(* Logix 5000 project; controller IOL_Sample vendor 1 type 14 code 196 rev 30.11; software revision 30.02; part 7 of 7 *)

TYPE Generic_16_Words :
STRUCT
   Data : INT[16];
END_STRUCT
END_TYPE

TYPE Generic_28_Bytes :
STRUCT
   Data : SINT[28];
END_STRUCT
END_TYPE

ADD_ON_INSTRUCTION Turck_TN_Q40   (* revision 1.0 *)
VAR_IN_OUT
   Process_Data_In : Generic_16_Words; {required}
   Process_Data_Out : Generic_16_Words; {required}
END_VAR
VAR_OUTPUT
   Ready_Flag : BOOL; {visible}   // 1 -> 0 or 0 -> 1: Command executed, new data available 0 or 1: No new data available
   Error : BOOL; {visible}   // 0: Command executed error-free 1: Command executed with error
   Tag : BOOL; {visible}   // 0: No tag within the detection range 1: Tag present at read/write head
   Antenna_State : BOOL; {visible}   // 0: RF field switched off 1: RF field switched on
   CMDCPY : SINT; {visible}   // Command Code Echo
   Error_Code : SINT; {visible}   // Error Code (Check Manual)
   ALR2 : BOOL; {visible}   // 0: Alarm 2 off 1: Alarm 2 on
   ALR1 : BOOL; {visible}   // 0: Alarm 1 off 1: Alarm 1 on
   Address : SINT; {visible}   // Address of the first memory block on the tag on which a command was executed
   RSSI : SINT; {visible}   // Signal Strength
END_VAR
VAR_IN_OUT
   Read_Data : Generic_28_Bytes; {required}   // Data read from Tag
END_VAR
VAR_INPUT
   Start : BOOL; {visible}   // 1 -> 0 or 0 -> 1: Execute command. The START bit switches status automatically with the automatic read and automatic write commands. 0 or 1: Idle
   N_Ant : BOOL; {visible}   // 0: Switch on RF field 1: Switch off RF field
   CMD : SINT; {visible}   // 0: No command 1: Automatic read 2: Automatic write 3: Read 4: Write 5: Display UID and time stamp
   NB_Block : SINT; {visible}   // Number of memory blocks to be read or written n EEPROM: max. 7 memory blocks n FRAM: max. 3 memory blocks
   Start_Address : INT; {visible}   // Address of the first memory block on the tag on which a command is to be executed
END_VAR
VAR_IN_OUT
   Write_Data : Generic_28_Bytes; {required}   // Data to write to Tag
END_VAR

ROUTINE Logic   (* ladder *)
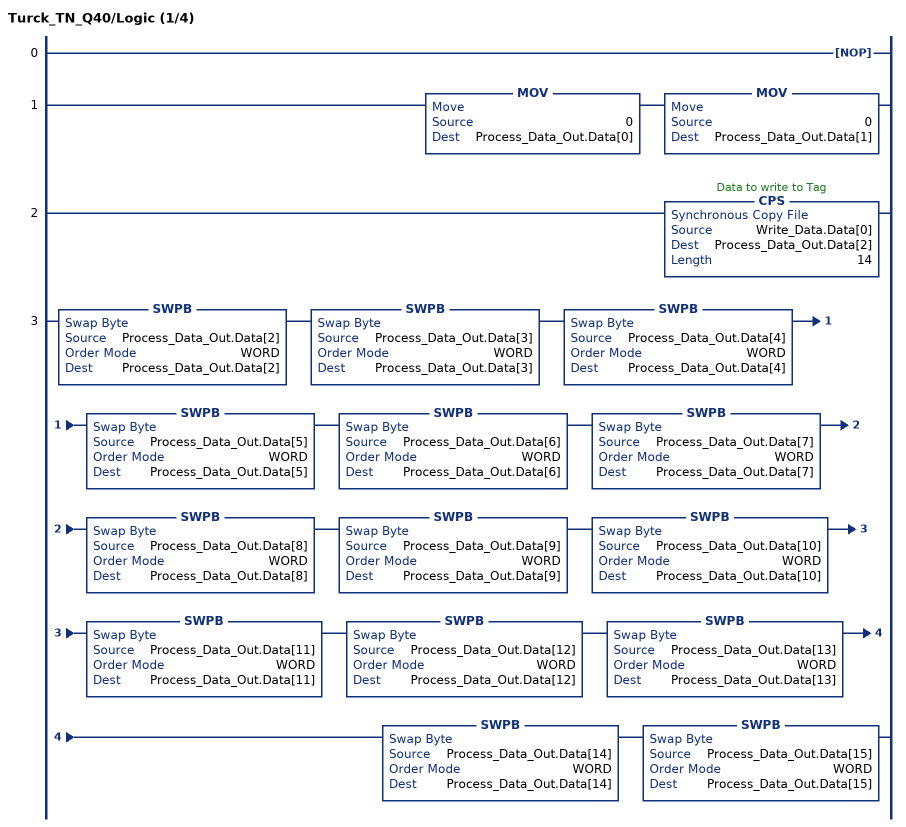
   0: NOP();
   1: MOV(0,Process_Data_Out.Data[0])MOV(0,Process_Data_Out.Data[1]);
   2: CPS(Write_Data.Data[0],Process_Data_Out.Data[2],14);
   3: SWPB(Process_Data_Out.Data[2],WORD,Process_Data_Out.Data[2])SWPB(Process_Data_Out.Data[3],WORD,Process_Data_Out.Data[3])SWPB(Process_Data_Out.Data[4],WORD,Process_Data_Out.Data[4])SWPB(Process_Data_Out.Data[5],WORD,Process_Data_Out.Data[5])SWPB(Process_Data_Out.Data[6],WORD,Process_Data_Out.Data[6])SWPB(Process_Data_Out.Data[7],WORD,Process_Data_Out.Data[7])SWPB(Process_Data_Out.Data[8],WORD,Process_Data_Out.Data[8])SWPB(Process_Data_Out.Data[9],WORD,Process_Data_Out.Data[9])SWPB(Process_Data_Out.Data[10],WORD,Process_Data_Out.Data[10])SWPB(Process_Data_Out.Data[11],WORD,Process_Data_Out.Data[11])SWPB(Process_Data_Out.Data[12],WORD,Process_Data_Out.Data[12])SWPB(Process_Data_Out.Data[13],WORD,Process_Data_Out.Data[13])SWPB(Process_Data_Out.Data[14],WORD,Process_Data_Out.Data[14])SWPB(Process_Data_Out.Data[15],WORD,Process_Data_Out.Data[15]);
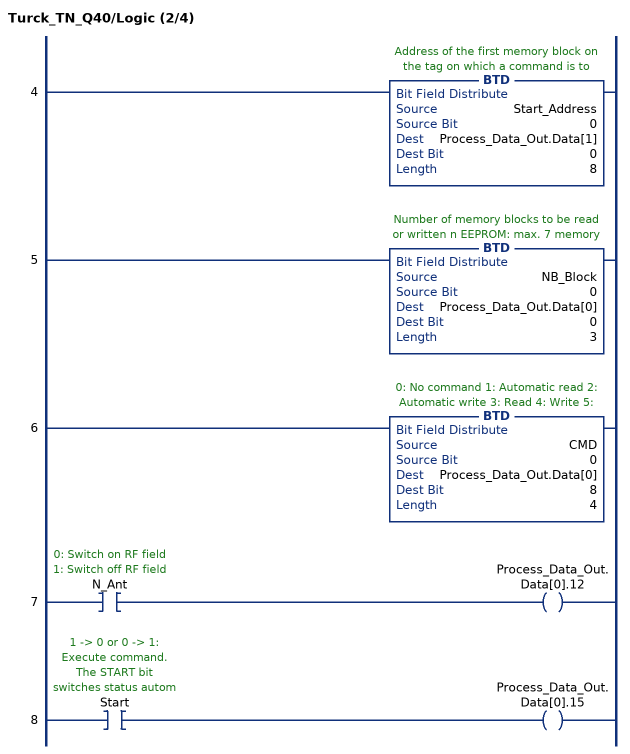
   4: BTD(Start_Address,0,Process_Data_Out.Data[1],0,8);
   5: BTD(NB_Block,0,Process_Data_Out.Data[0],0,3);
   6: BTD(CMD,0,Process_Data_Out.Data[0],8,4);
   7: XIC(N_Ant)OTE(Process_Data_Out.Data[0].12);
   8: XIC(Start)OTE(Process_Data_Out.Data[0].15);
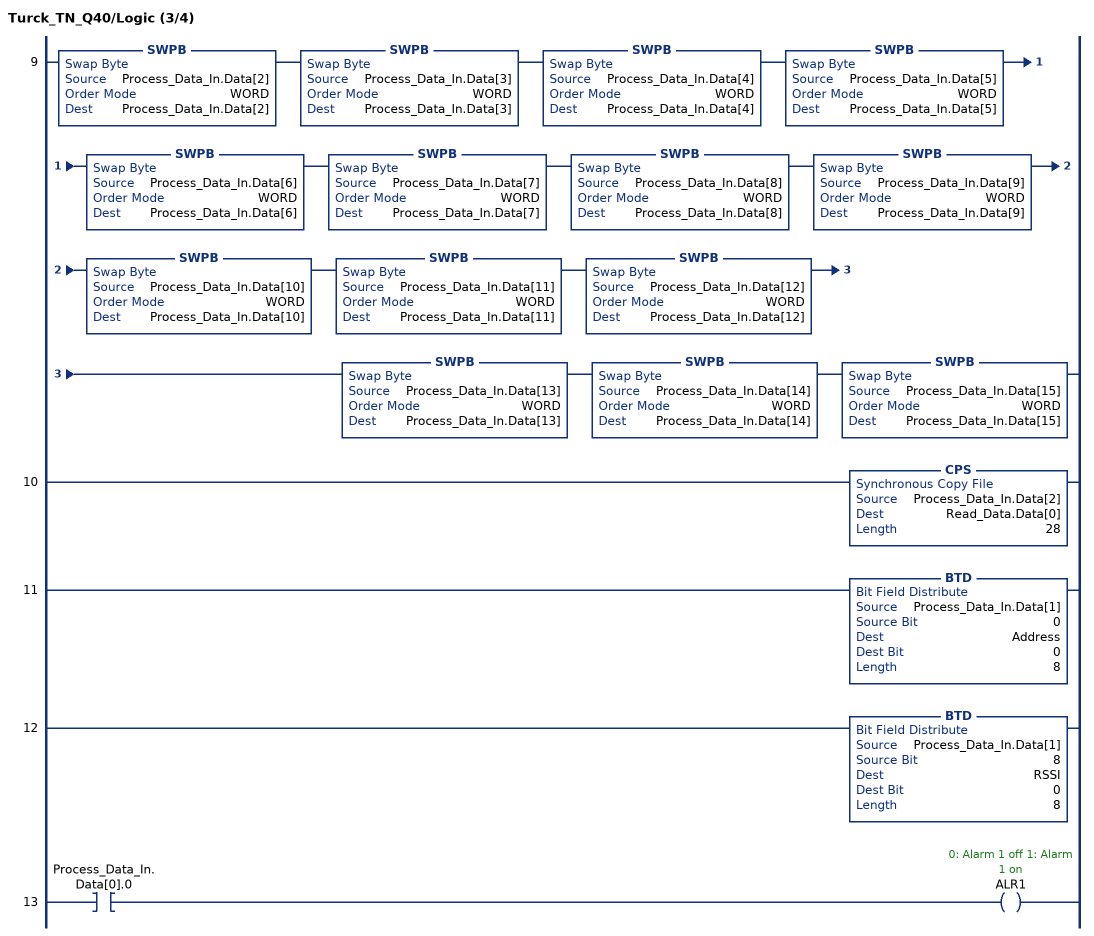
   9: SWPB(Process_Data_In.Data[2],WORD,Process_Data_In.Data[2])SWPB(Process_Data_In.Data[3],WORD,Process_Data_In.Data[3])SWPB(Process_Data_In.Data[4],WORD,Process_Data_In.Data[4])SWPB(Process_Data_In.Data[5],WORD,Process_Data_In.Data[5])SWPB(Process_Data_In.Data[6],WORD,Process_Data_In.Data[6])SWPB(Process_Data_In.Data[7],WORD,Process_Data_In.Data[7])SWPB(Process_Data_In.Data[8],WORD,Process_Data_In.Data[8])SWPB(Process_Data_In.Data[9],WORD,Process_Data_In.Data[9])SWPB(Process_Data_In.Data[10],WORD,Process_Data_In.Data[10])SWPB(Process_Data_In.Data[11],WORD,Process_Data_In.Data[11])SWPB(Process_Data_In.Data[12],WORD,Process_Data_In.Data[12])SWPB(Process_Data_In.Data[13],WORD,Process_Data_In.Data[13])SWPB(Process_Data_In.Data[14],WORD,Process_Data_In.Data[14])SWPB(Process_Data_In.Data[15],WORD,Process_Data_In.Data[15]);
   10: CPS(Process_Data_In.Data[2],Read_Data.Data[0],28);
   11: BTD(Process_Data_In.Data[1],0,Address,0,8);
   12: BTD(Process_Data_In.Data[1],8,RSSI,0,8);
   13: XIC(Process_Data_In.Data[0].0)OTE(ALR1);
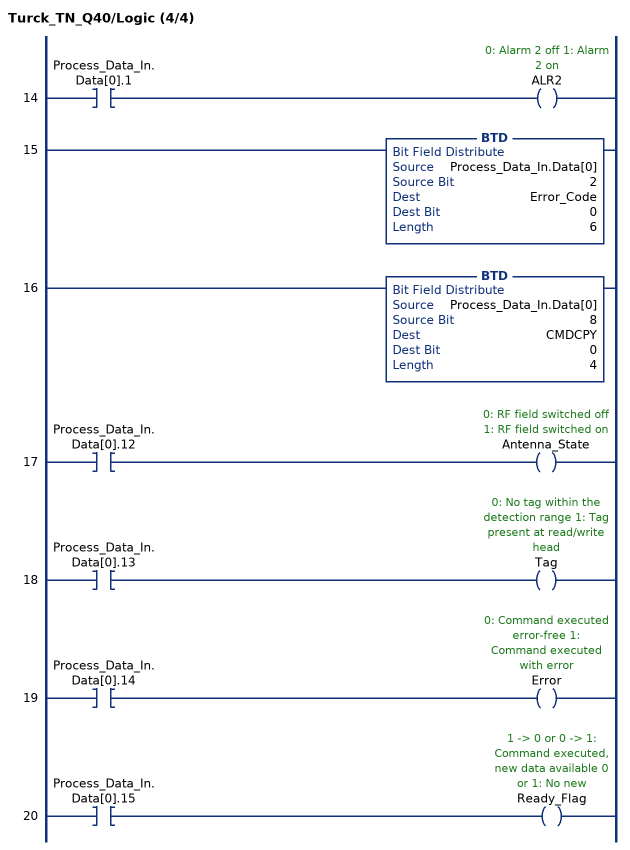
   14: XIC(Process_Data_In.Data[0].1)OTE(ALR2);
   15: BTD(Process_Data_In.Data[0],2,Error_Code,0,6);
   16: BTD(Process_Data_In.Data[0],8,CMDCPY,0,4);
   17: XIC(Process_Data_In.Data[0].12)OTE(Antenna_State);
   18: XIC(Process_Data_In.Data[0].13)OTE(Tag);
   19: XIC(Process_Data_In.Data[0].14)OTE(Error);
   20: XIC(Process_Data_In.Data[0].15)OTE(Ready_Flag);
END_ROUTINE
END_ADD_ON_INSTRUCTION

VAR_GLOBAL   (* controller tags *)
   Q40 : Turck_TN_Q40 := (Ready_Flag := 1, Antenna_State := 1, CMDCPY := 3, Start := 1, CMD := 3, NB_Block := 7);   // RFID Interface: Command and Status
   Q40_PD0 : Generic_16_Words := (Data[0] := -31993, Data[2] := 258, Data[3] := 772, Data[4] := 1286, Data[5] := 1800, Data[6] := 2314, Data[7] := 2828, Data[8] := 3342, Data[9] := 3856, Data[10] := 4370, Data[11] := 4884, Data[12] := 5398, Data[13] := 5912, Data[14] := 6426, Data[15] := 6940);
   Q40_Process_Data : Generic_16_Words := (Data[0] := -27904, Data[2] := 513, Data[3] := 1027, Data[4] := 1541, Data[5] := 2055, Data[6] := 2569, Data[7] := 3083, Data[8] := 3597, Data[9] := 4111, Data[10] := 4625, Data[11] := 5139, Data[12] := 5653, Data[13] := 6167, Data[14] := 6681, Data[15] := 7195);
   Q40_Read_Data_Buffer : Generic_28_Bytes := (Data[0] := 1, Data[1] := 2, Data[2] := 3, Data[3] := 4, Data[4] := 5, Data[5] := 6, Data[6] := 7, Data[7] := 8, Data[8] := 9, Data[9] := 10, Data[10] := 11, Data[11] := 12, Data[12] := 13, Data[13] := 14, Data[14] := 15, Data[15] := 16, Data[16] := 17, Data[17] := 18, Data[18] := 19, Data[19] := 20, Data[20] := 21, Data[21] := 22, Data[22] := 23, Data[23] := 24, Data[24] := 25, Data[25] := 26, Data[26] := 27, Data[27] := 28);   // Read Data Buffer
        .Data[0]   // Station Status Word
        .Data[0].0   // Module Diagnostics Available
        .Data[0].1   // Reserved
        .Data[0].2   // Reserved
        .Data[0].3   // Reserved
        .Data[0].4   // Reserved
        .Data[0].5   // Reserved
        .Data[0].6   // Reserved
        .Data[0].7   // Undervoltage Field Supply V2
        .Data[1]   // DI input, Input value
        .Data[1].0   // IOL 0 - DI input (ENUM bit0): 0=off, 1=on
        .Data[1].1   // DXP 1 - Input value (ENUM bit0): 0=off, 1=on
        .Data[1].2   // IOL 2 - DI input (ENUM bit0): 0=off, 1=on
        .Data[1].3   // DXP 3 - Input value (ENUM bit0): 0=off, 1=on
        .Data[1].4   // IOL 4 - DI input (ENUM bit0): 0=off, 1=on
        .Data[1].5   // DXP 5 - Input value (ENUM bit0): 0=off, 1=on
        .Data[1].6   // IOL 6 - DI input (ENUM bit0): 0=off, 1=on
        .Data[1].7   // DXP 7 - Input value (ENUM bit0): 0=off, 1=on
        .Data[2]   // Input values valid
        .Data[2].0   // IOL 0 - Input values valid (ENUM bit0): 0=no, 1=yes
        .Data[2].1   // Reserved
        .Data[2].2   // IOL 2 - Input values valid (ENUM bit0): 0=no, 1=yes
        .Data[2].3   // Reserved
        .Data[2].4   // IOL 4 - Input values valid (ENUM bit0): 0=no, 1=yes
        .Data[2].5   // Reserved
        .Data[2].6   // IOL 6 - Input values valid (ENUM bit0): 0=no, 1=yes
        .Data[2].7   // Reserved
        .Data[3]   // IO-Link Port 1 - Input data word 0
        .Data[3].0   // IO-Link Port 1 - Input data word 0 (INT bit0)
        .Data[3].1   // IO-Link Port 1 - Input data word 0 (INT bit1)
        .Data[3].2   // IO-Link Port 1 - Input data word 0 (INT bit2)
        .Data[3].3   // IO-Link Port 1 - Input data word 0 (INT bit3)
        .Data[3].4   // IO-Link Port 1 - Input data word 0 (INT bit4)
        .Data[3].5   // IO-Link Port 1 - Input data word 0 (INT bit5)
        .Data[3].6   // IO-Link Port 1 - Input data word 0 (INT bit6)
        .Data[3].7   // IO-Link Port 1 - Input data word 0 (INT bit7)
        .Data[4]   // IO-Link Port 1 - Input data word 1
        .Data[4].0   // IO-Link Port 1 - Input data word 1 (INT bit0)
        .Data[4].1   // IO-Link Port 1 - Input data word 1 (INT bit1)
        .Data[4].2   // IO-Link Port 1 - Input data word 1 (INT bit2)
        .Data[4].3   // IO-Link Port 1 - Input data word 1 (INT bit3)
        .Data[4].4   // IO-Link Port 1 - Input data word 1 (INT bit4)
        .Data[4].5   // IO-Link Port 1 - Input data word 1 (INT bit5)
        .Data[4].6   // IO-Link Port 1 - Input data word 1 (INT bit6)
        .Data[4].7   // IO-Link Port 1 - Input data word 1 (INT bit7)
        .Data[5]   // IO-Link Port 1 - Input data word 2
        .Data[5].0   // IO-Link Port 1 - Input data word 2 (INT bit0)
        .Data[5].1   // IO-Link Port 1 - Input data word 2 (INT bit1)
        .Data[5].2   // IO-Link Port 1 - Input data word 2 (INT bit2)
        .Data[5].3   // IO-Link Port 1 - Input data word 2 (INT bit3)
        .Data[5].4   // IO-Link Port 1 - Input data word 2 (INT bit4)
        .Data[5].5   // IO-Link Port 1 - Input data word 2 (INT bit5)
        .Data[5].6   // IO-Link Port 1 - Input data word 2 (INT bit6)
        .Data[5].7   // IO-Link Port 1 - Input data word 2 (INT bit7)
        .Data[6]   // IO-Link Port 1 - Input data word 3
        .Data[6].0   // IO-Link Port 1 - Input data word 3 (INT bit0)
        .Data[6].1   // IO-Link Port 1 - Input data word 3 (INT bit1)
        .Data[6].2   // IO-Link Port 1 - Input data word 3 (INT bit2)
        .Data[6].3   // IO-Link Port 1 - Input data word 3 (INT bit3)
        .Data[6].4   // IO-Link Port 1 - Input data word 3 (INT bit4)
        .Data[6].5   // IO-Link Port 1 - Input data word 3 (INT bit5)
        .Data[6].6   // IO-Link Port 1 - Input data word 3 (INT bit6)
        .Data[6].7   // IO-Link Port 1 - Input data word 3 (INT bit7)
        .Data[7]   // IO-Link Port 1 - Input data word 4
        .Data[7].0   // IO-Link Port 1 - Input data word 4 (INT bit0)
        .Data[7].1   // IO-Link Port 1 - Input data word 4 (INT bit1)
        .Data[7].2   // IO-Link Port 1 - Input data word 4 (INT bit2)
        .Data[7].3   // IO-Link Port 1 - Input data word 4 (INT bit3)
        .Data[7].4   // IO-Link Port 1 - Input data word 4 (INT bit4)
        .Data[7].5   // IO-Link Port 1 - Input data word 4 (INT bit5)
        .Data[7].6   // IO-Link Port 1 - Input data word 4 (INT bit6)
        .Data[7].7   // IO-Link Port 1 - Input data word 4 (INT bit7)
        .Data[8]   // IO-Link Port 1 - Input data word 5
        .Data[8].0   // IO-Link Port 1 - Input data word 5 (INT bit0)
        .Data[8].1   // IO-Link Port 1 - Input data word 5 (INT bit1)
        .Data[8].2   // IO-Link Port 1 - Input data word 5 (INT bit2)
        .Data[8].3   // IO-Link Port 1 - Input data word 5 (INT bit3)
        .Data[8].4   // IO-Link Port 1 - Input data word 5 (INT bit4)
        .Data[8].5   // IO-Link Port 1 - Input data word 5 (INT bit5)
        .Data[8].6   // IO-Link Port 1 - Input data word 5 (INT bit6)
        .Data[8].7   // IO-Link Port 1 - Input data word 5 (INT bit7)
        .Data[9]   // IO-Link Port 1 - Input data word 6
        .Data[9].0   // IO-Link Port 1 - Input data word 6 (INT bit0)
        .Data[9].1   // IO-Link Port 1 - Input data word 6 (INT bit1)
        .Data[9].2   // IO-Link Port 1 - Input data word 6 (INT bit2)
        .Data[9].3   // IO-Link Port 1 - Input data word 6 (INT bit3)
        .Data[9].4   // IO-Link Port 1 - Input data word 6 (INT bit4)
        .Data[9].5   // IO-Link Port 1 - Input data word 6 (INT bit5)
        .Data[9].6   // IO-Link Port 1 - Input data word 6 (INT bit6)
        .Data[9].7   // IO-Link Port 1 - Input data word 6 (INT bit7)
        .Data[10]   // IO-Link Port 1 - Input data word 7
        .Data[10].0   // IO-Link Port 1 - Input data word 7 (INT bit0)
        .Data[10].1   // IO-Link Port 1 - Input data word 7 (INT bit1)
        .Data[10].2   // IO-Link Port 1 - Input data word 7 (INT bit2)
        .Data[10].3   // IO-Link Port 1 - Input data word 7 (INT bit3)
        .Data[10].4   // IO-Link Port 1 - Input data word 7 (INT bit4)
        .Data[10].5   // IO-Link Port 1 - Input data word 7 (INT bit5)
        .Data[10].6   // IO-Link Port 1 - Input data word 7 (INT bit6)
        .Data[10].7   // IO-Link Port 1 - Input data word 7 (INT bit7)
        .Data[11]   // IO-Link Port 1 - Input data word 8
        .Data[11].0   // IO-Link Port 1 - Input data word 8 (INT bit0)
        .Data[11].1   // IO-Link Port 1 - Input data word 8 (INT bit1)
        .Data[11].2   // IO-Link Port 1 - Input data word 8 (INT bit2)
        .Data[11].3   // IO-Link Port 1 - Input data word 8 (INT bit3)
        .Data[11].4   // IO-Link Port 1 - Input data word 8 (INT bit4)
        .Data[11].5   // IO-Link Port 1 - Input data word 8 (INT bit5)
        .Data[11].6   // IO-Link Port 1 - Input data word 8 (INT bit6)
        .Data[11].7   // IO-Link Port 1 - Input data word 8 (INT bit7)
        .Data[12]   // IO-Link Port 1 - Input data word 9
        .Data[12].0   // IO-Link Port 1 - Input data word 9 (INT bit0)
        .Data[12].1   // IO-Link Port 1 - Input data word 9 (INT bit1)
        .Data[12].2   // IO-Link Port 1 - Input data word 9 (INT bit2)
        .Data[12].3   // IO-Link Port 1 - Input data word 9 (INT bit3)
        .Data[12].4   // IO-Link Port 1 - Input data word 9 (INT bit4)
        .Data[12].5   // IO-Link Port 1 - Input data word 9 (INT bit5)
        .Data[12].6   // IO-Link Port 1 - Input data word 9 (INT bit6)
        .Data[12].7   // IO-Link Port 1 - Input data word 9 (INT bit7)
        .Data[13]   // IO-Link Port 1 - Input data word 10
        .Data[13].0   // IO-Link Port 1 - Input data word 10 (INT bit0)
        .Data[13].1   // IO-Link Port 1 - Input data word 10 (INT bit1)
        .Data[13].2   // IO-Link Port 1 - Input data word 10 (INT bit2)
        .Data[13].3   // IO-Link Port 1 - Input data word 10 (INT bit3)
        .Data[13].4   // IO-Link Port 1 - Input data word 10 (INT bit4)
        .Data[13].5   // IO-Link Port 1 - Input data word 10 (INT bit5)
        .Data[13].6   // IO-Link Port 1 - Input data word 10 (INT bit6)
        .Data[13].7   // IO-Link Port 1 - Input data word 10 (INT bit7)
        .Data[14]   // IO-Link Port 1 - Input data word 11
        .Data[14].0   // IO-Link Port 1 - Input data word 11 (INT bit0)
        .Data[14].1   // IO-Link Port 1 - Input data word 11 (INT bit1)
        .Data[14].2   // IO-Link Port 1 - Input data word 11 (INT bit2)
        .Data[14].3   // IO-Link Port 1 - Input data word 11 (INT bit3)
        .Data[14].4   // IO-Link Port 1 - Input data word 11 (INT bit4)
        .Data[14].5   // IO-Link Port 1 - Input data word 11 (INT bit5)
        .Data[14].6   // IO-Link Port 1 - Input data word 11 (INT bit6)
        .Data[14].7   // IO-Link Port 1 - Input data word 11 (INT bit7)
        .Data[15]   // IO-Link Port 1 - Input data word 12
        .Data[15].0   // IO-Link Port 1 - Input data word 12 (INT bit0)
        .Data[15].1   // IO-Link Port 1 - Input data word 12 (INT bit1)
        .Data[15].2   // IO-Link Port 1 - Input data word 12 (INT bit2)
        .Data[15].3   // IO-Link Port 1 - Input data word 12 (INT bit3)
        .Data[15].4   // IO-Link Port 1 - Input data word 12 (INT bit4)
        .Data[15].5   // IO-Link Port 1 - Input data word 12 (INT bit5)
        .Data[15].6   // IO-Link Port 1 - Input data word 12 (INT bit6)
        .Data[15].7   // IO-Link Port 1 - Input data word 12 (INT bit7)
        .Data[16]   // IO-Link Port 1 - Input data word 13
        .Data[16].0   // IO-Link Port 1 - Input data word 13 (INT bit0)
        .Data[16].1   // IO-Link Port 1 - Input data word 13 (INT bit1)
        .Data[16].2   // IO-Link Port 1 - Input data word 13 (INT bit2)
        .Data[16].3   // IO-Link Port 1 - Input data word 13 (INT bit3)
        .Data[16].4   // IO-Link Port 1 - Input data word 13 (INT bit4)
        .Data[16].5   // IO-Link Port 1 - Input data word 13 (INT bit5)
        .Data[16].6   // IO-Link Port 1 - Input data word 13 (INT bit6)
        .Data[16].7   // IO-Link Port 1 - Input data word 13 (INT bit7)
        .Data[17]   // IO-Link Port 1 - Input data word 14
        .Data[17].0   // IO-Link Port 1 - Input data word 14 (INT bit0)
        .Data[17].1   // IO-Link Port 1 - Input data word 14 (INT bit1)
        .Data[17].2   // IO-Link Port 1 - Input data word 14 (INT bit2)
        .Data[17].3   // IO-Link Port 1 - Input data word 14 (INT bit3)
        .Data[17].4   // IO-Link Port 1 - Input data word 14 (INT bit4)
        .Data[17].5   // IO-Link Port 1 - Input data word 14 (INT bit5)
        .Data[17].6   // IO-Link Port 1 - Input data word 14 (INT bit6)
        .Data[17].7   // IO-Link Port 1 - Input data word 14 (INT bit7)
        .Data[18]   // IO-Link Port 1 - Input data word 15
        .Data[18].0   // IO-Link Port 1 - Input data word 15 (INT bit0)
        .Data[18].1   // IO-Link Port 1 - Input data word 15 (INT bit1)
        .Data[18].2   // IO-Link Port 1 - Input data word 15 (INT bit2)
        .Data[18].3   // IO-Link Port 1 - Input data word 15 (INT bit3)
        .Data[18].4   // IO-Link Port 1 - Input data word 15 (INT bit4)
        .Data[18].5   // IO-Link Port 1 - Input data word 15 (INT bit5)
        .Data[18].6   // IO-Link Port 1 - Input data word 15 (INT bit6)
        .Data[18].7   // IO-Link Port 1 - Input data word 15 (INT bit7)
        .Data[19]   // IO-Link Port 2 - Input data word 0
        .Data[19].0   // IO-Link Port 2 - Input data word 0 (INT bit0)
        .Data[19].1   // IO-Link Port 2 - Input data word 0 (INT bit1)
        .Data[19].2   // IO-Link Port 2 - Input data word 0 (INT bit2)
        .Data[19].3   // IO-Link Port 2 - Input data word 0 (INT bit3)
        .Data[19].4   // IO-Link Port 2 - Input data word 0 (INT bit4)
        .Data[19].5   // IO-Link Port 2 - Input data word 0 (INT bit5)
        .Data[19].6   // IO-Link Port 2 - Input data word 0 (INT bit6)
        .Data[19].7   // IO-Link Port 2 - Input data word 0 (INT bit7)
        .Data[20]   // IO-Link Port 2 - Input data word 1
        .Data[20].0   // IO-Link Port 2 - Input data word 1 (INT bit0)
        .Data[20].1   // IO-Link Port 2 - Input data word 1 (INT bit1)
        .Data[20].2   // IO-Link Port 2 - Input data word 1 (INT bit2)
        .Data[20].3   // IO-Link Port 2 - Input data word 1 (INT bit3)
        .Data[20].4   // IO-Link Port 2 - Input data word 1 (INT bit4)
        .Data[20].5   // IO-Link Port 2 - Input data word 1 (INT bit5)
        .Data[20].6   // IO-Link Port 2 - Input data word 1 (INT bit6)
        .Data[20].7   // IO-Link Port 2 - Input data word 1 (INT bit7)
        .Data[21]   // IO-Link Port 2 - Input data word 2
        .Data[21].0   // IO-Link Port 2 - Input data word 2 (INT bit0)
        .Data[21].1   // IO-Link Port 2 - Input data word 2 (INT bit1)
        .Data[21].2   // IO-Link Port 2 - Input data word 2 (INT bit2)
        .Data[21].3   // IO-Link Port 2 - Input data word 2 (INT bit3)
        .Data[21].4   // IO-Link Port 2 - Input data word 2 (INT bit4)
        .Data[21].5   // IO-Link Port 2 - Input data word 2 (INT bit5)
        .Data[21].6   // IO-Link Port 2 - Input data word 2 (INT bit6)
        .Data[21].7   // IO-Link Port 2 - Input data word 2 (INT bit7)
        .Data[22]   // IO-Link Port 2 - Input data word 3
        .Data[22].0   // IO-Link Port 2 - Input data word 3 (INT bit0)
        .Data[22].1   // IO-Link Port 2 - Input data word 3 (INT bit1)
        .Data[22].2   // IO-Link Port 2 - Input data word 3 (INT bit2)
        .Data[22].3   // IO-Link Port 2 - Input data word 3 (INT bit3)
        .Data[22].4   // IO-Link Port 2 - Input data word 3 (INT bit4)
        .Data[22].5   // IO-Link Port 2 - Input data word 3 (INT bit5)
        .Data[22].6   // IO-Link Port 2 - Input data word 3 (INT bit6)
        .Data[22].7   // IO-Link Port 2 - Input data word 3 (INT bit7)
        .Data[23]   // IO-Link Port 2 - Input data word 4
        .Data[23].0   // IO-Link Port 2 - Input data word 4 (INT bit0)
        .Data[23].1   // IO-Link Port 2 - Input data word 4 (INT bit1)
        .Data[23].2   // IO-Link Port 2 - Input data word 4 (INT bit2)
        .Data[23].3   // IO-Link Port 2 - Input data word 4 (INT bit3)
        .Data[23].4   // IO-Link Port 2 - Input data word 4 (INT bit4)
        .Data[23].5   // IO-Link Port 2 - Input data word 4 (INT bit5)
        .Data[23].6   // IO-Link Port 2 - Input data word 4 (INT bit6)
        .Data[23].7   // IO-Link Port 2 - Input data word 4 (INT bit7)
        .Data[24]   // IO-Link Port 2 - Input data word 5
        .Data[24].0   // IO-Link Port 2 - Input data word 5 (INT bit0)
        .Data[24].1   // IO-Link Port 2 - Input data word 5 (INT bit1)
        .Data[24].2   // IO-Link Port 2 - Input data word 5 (INT bit2)
        .Data[24].3   // IO-Link Port 2 - Input data word 5 (INT bit3)
        .Data[24].4   // IO-Link Port 2 - Input data word 5 (INT bit4)
        .Data[24].5   // IO-Link Port 2 - Input data word 5 (INT bit5)
        .Data[24].6   // IO-Link Port 2 - Input data word 5 (INT bit6)
        .Data[24].7   // IO-Link Port 2 - Input data word 5 (INT bit7)
        .Data[25]   // IO-Link Port 2 - Input data word 6
        .Data[25].0   // IO-Link Port 2 - Input data word 6 (INT bit0)
        .Data[25].1   // IO-Link Port 2 - Input data word 6 (INT bit1)
        .Data[25].2   // IO-Link Port 2 - Input data word 6 (INT bit2)
        .Data[25].3   // IO-Link Port 2 - Input data word 6 (INT bit3)
        .Data[25].4   // IO-Link Port 2 - Input data word 6 (INT bit4)
        .Data[25].5   // IO-Link Port 2 - Input data word 6 (INT bit5)
        .Data[25].6   // IO-Link Port 2 - Input data word 6 (INT bit6)
        .Data[25].7   // IO-Link Port 2 - Input data word 6 (INT bit7)
        .Data[26]   // IO-Link Port 2 - Input data word 7
        .Data[26].0   // IO-Link Port 2 - Input data word 7 (INT bit0)
        .Data[26].1   // IO-Link Port 2 - Input data word 7 (INT bit1)
        .Data[26].2   // IO-Link Port 2 - Input data word 7 (INT bit2)
        .Data[26].3   // IO-Link Port 2 - Input data word 7 (INT bit3)
        .Data[26].4   // IO-Link Port 2 - Input data word 7 (INT bit4)
        .Data[26].5   // IO-Link Port 2 - Input data word 7 (INT bit5)
        .Data[26].6   // IO-Link Port 2 - Input data word 7 (INT bit6)
        .Data[26].7   // IO-Link Port 2 - Input data word 7 (INT bit7)
        .Data[27]   // IO-Link Port 2 - Input data word 8
        .Data[27].0   // IO-Link Port 2 - Input data word 8 (INT bit0)
        .Data[27].1   // IO-Link Port 2 - Input data word 8 (INT bit1)
        .Data[27].2   // IO-Link Port 2 - Input data word 8 (INT bit2)
        .Data[27].3   // IO-Link Port 2 - Input data word 8 (INT bit3)
        .Data[27].4   // IO-Link Port 2 - Input data word 8 (INT bit4)
        .Data[27].5   // IO-Link Port 2 - Input data word 8 (INT bit5)
        .Data[27].6   // IO-Link Port 2 - Input data word 8 (INT bit6)
        .Data[27].7   // IO-Link Port 2 - Input data word 8 (INT bit7)
   Q40_Write_Data_Buffer : Generic_28_Bytes;   // Write Data Buffer
END_VAR

PROGRAM MainProgram   (* main routine MainRoutine *)

ROUTINE MainRoutine   (* ladder *)
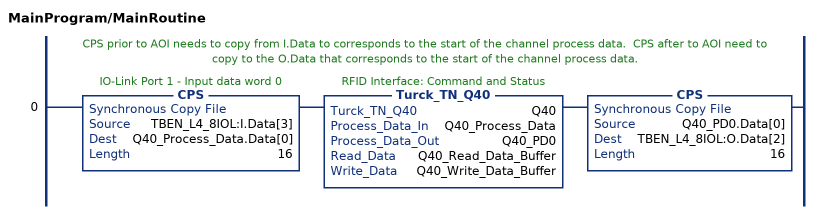
   // CPS prior to AOI needs to copy from I.Data to corresponds to the start of the channel process data.  CPS after to AOI need to copy to the O.Data that corresponds to the start of the channel process data.
   0: CPS(TBEN_L4_8IOL:I.Data[3],Q40_Process_Data.Data[0],16)Turck_TN_Q40(Q40,Q40_Process_Data,Q40_PD0,Q40_Read_Data_Buffer,Q40_Write_Data_Buffer)CPS(Q40_PD0.Data[0],TBEN_L4_8IOL:O.Data[2],16);
END_ROUTINE
END_PROGRAM
